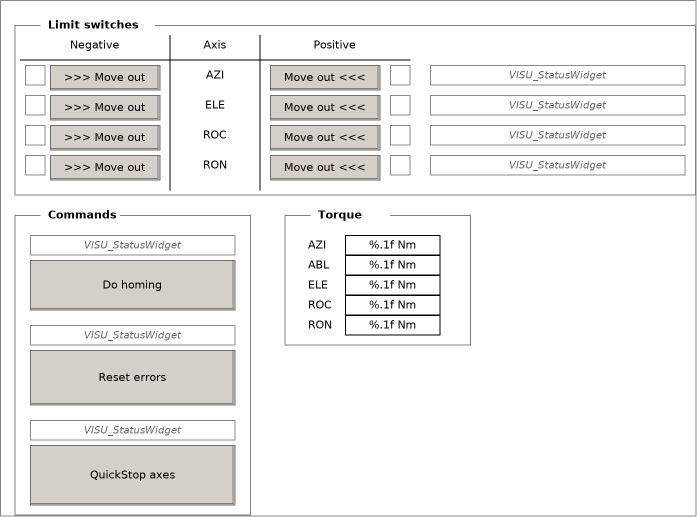
VISUALIZATION VISU_AxesAdvanced  // 697x517
VAR_IN_OUT
	ref : Axes;
    widget : AxesWidget;
END_VAR
    Polyline (120,215) (250,215) (250,515) (15,515) (15,215) (40,215)
    Polyline (155,25) (695,25) (695,195) (15,195) (15,25) (40,25)
    Label (45,15 100x20), "Limit switches"
    Label (170,60 90x30), "AZI"
    Frame (390,65 20x20)
        shows VISU_State_gray_red(state := ref.parts.azi.positiveLimitSwitchError)
    Line (260,190) (260,35)
    Line (170,190) (170,35)
    Label (260,30 150x30), "Positive"
    Label (20,30 150x30), "Negative"
    Line (410,60) (20,60)
    Label (170,30 90x30), "Axis"
    Button (270,65 110x25), "Move out <<<", input disabled if: ref.parts.azi.processes.moveOutOfLimitSwitch.statuses.enabledStatus.disabled
        OnMouseClick: execute { ref.parts.azi.processes.moveOutOfLimitSwitch.set.switch := LimitSwitches.POSITIVE_LIMIT_SWITCH; ref.parts.azi.processes.moveOutOfLimitSwitch.do_request := TRUE; }
    Frame (25,65 20x20)
        shows VISU_State_gray_red(state := ref.parts.azi.negativeLimitSwitchError)
    Button (50,65 110x25), ">>> Move out", input disabled if: ref.parts.azi.processes.moveOutOfLimitSwitch.statuses.enabledStatus.disabled
        OnMouseClick: execute { ref.parts.azi.processes.moveOutOfLimitSwitch.set.switch := LimitSwitches.NEGATIVE_LIMIT_SWITCH; ref.parts.azi.processes.moveOutOfLimitSwitch.do_request := TRUE; }
    Label (170,90 90x30), "ELE"
    Frame (390,95 20x20)
        shows VISU_State_gray_red(state := ref.parts.ele.positiveLimitSwitchError)
    Button (270,95 110x25), "Move out <<<", input disabled if: ref.parts.ele.processes.moveOutOfLimitSwitch.statuses.enabledStatus.disabled
        OnMouseClick: execute { ref.parts.ele.processes.moveOutOfLimitSwitch.set.switch := LimitSwitches.POSITIVE_LIMIT_SWITCH; ref.parts.ele.processes.moveOutOfLimitSwitch.do_request := TRUE; }
    Frame (25,95 20x20)
        shows VISU_State_gray_red(state := ref.parts.ele.negativeLimitSwitchError)
    Button (50,95 110x25), ">>> Move out", input disabled if: ref.parts.ele.processes.moveOutOfLimitSwitch.statuses.enabledStatus.disabled
        OnMouseClick: execute { ref.parts.ele.processes.moveOutOfLimitSwitch.set.switch := LimitSwitches.NEGATIVE_LIMIT_SWITCH; ref.parts.ele.processes.moveOutOfLimitSwitch.do_request := TRUE; }
    Label (170,120 90x30), "ROC"
    Frame (390,125 20x20)
        shows VISU_State_gray_red(state := ref.parts.roc.positiveLimitSwitchError)
    Button (270,125 110x25), "Move out <<<", input disabled if: ref.parts.roc.processes.moveOutOfLimitSwitch.statuses.enabledStatus.disabled
        OnMouseClick: execute { ref.parts.roc.processes.moveOutOfLimitSwitch.set.switch := LimitSwitches.POSITIVE_LIMIT_SWITCH; ref.parts.roc.processes.moveOutOfLimitSwitch.do_request := TRUE; }
    Frame (25,125 20x20)
        shows VISU_State_gray_red(state := ref.parts.roc.negativeLimitSwitchError)
    Button (50,125 110x25), ">>> Move out", input disabled if: ref.parts.roc.processes.moveOutOfLimitSwitch.statuses.enabledStatus.disabled
        OnMouseClick: execute { ref.parts.roc.processes.moveOutOfLimitSwitch.set.switch := LimitSwitches.NEGATIVE_LIMIT_SWITCH; ref.parts.roc.processes.moveOutOfLimitSwitch.do_request := TRUE; }
    Label (170,150 90x30), "RON"
    Frame (390,155 20x20)
        shows VISU_State_gray_red(state := ref.parts.ron.positiveLimitSwitchError)
    Button (270,155 110x25), "Move out <<<", input disabled if: ref.parts.ron.processes.moveOutOfLimitSwitch.statuses.enabledStatus.disabled
        OnMouseClick: execute { ref.parts.ron.processes.moveOutOfLimitSwitch.set.switch := LimitSwitches.POSITIVE_LIMIT_SWITCH; ref.parts.ron.processes.moveOutOfLimitSwitch.do_request := TRUE; }
    Frame (25,155 20x20)
        shows VISU_State_gray_red(state := ref.parts.ron.negativeLimitSwitchError)
    Button (50,155 110x25), ">>> Move out", input disabled if: ref.parts.ron.processes.moveOutOfLimitSwitch.statuses.enabledStatus.disabled
        OnMouseClick: execute { ref.parts.ron.processes.moveOutOfLimitSwitch.set.switch := LimitSwitches.NEGATIVE_LIMIT_SWITCH; ref.parts.ron.processes.moveOutOfLimitSwitch.do_request := TRUE; }
    Frame (430,65 255x20)
        shows VISU_StatusWidget(widget := widget.axes.azi.processes_moveOutOfLimitSwitchStatus)
    Frame (430,95 255x20)
        shows VISU_StatusWidget(widget := widget.axes.ele.processes_moveOutOfLimitSwitchStatus)
    Frame (430,125 255x20)
        shows VISU_StatusWidget(widget := widget.axes.roc.processes_moveOutOfLimitSwitchStatus)
    Frame (430,155 255x20)
        shows VISU_StatusWidget(widget := widget.axes.ron.processes_moveOutOfLimitSwitchStatus)
    Button (30,260 205x50), "Do homing", input disabled if: ref.processes.doHoming.statuses.enabledStatus.disabled
        OnMouseClick: execute { ref.processes.doHoming.do_request := TRUE; }
    Label (45,205 85x20), "Commands"
    Button (30,350 205x55), "Reset errors", input disabled if: ref.processes.reset.statuses.enabledStatus.disabled
        OnMouseClick: execute { ref.processes.reset.do_request := TRUE; }
    Frame (30,325 205x20)
        shows VISU_StatusWidget(widget := widget.processes_resetStatus)
        p4168582468: ref.processes.reset.actualStatus
    Frame (30,235 205x20)
        shows VISU_StatusWidget(widget := widget.processes_doHomingStatus)
        p4168582468: ref.processes.doHoming.actualStatus
    Button (30,445 205x60), "QuickStop axes", input disabled if: ref.processes.quickStop.statuses.enabledStatus.disabled
        OnMouseClick: execute { ref.processes.quickStop.do_request := TRUE; }
    Frame (30,420 205x20)
        shows VISU_StatusWidget(widget := widget.processes_quickStopStatus)
        p4168582468: ref.processes.quickStop.actualStatus
    Label (305,235 40x20), "AZI"
    Rectangle (345,235 95x20), "%.1f Nm", text variable: ref.parts.azi.actTorqueAzi.newtonmeter.value
    Label (305,255 40x20), "ABL"
    Rectangle (345,255 95x20), "%.1f Nm", text variable: ref.parts.azi.actTorqueAbl.newtonmeter.value
    Label (305,275 40x20), "ELE"
    Rectangle (345,275 95x20), "%.1f Nm", text variable: ref.parts.ele.actTorque.newtonmeter.value
    Label (305,295 40x20), "ROC"
    Rectangle (345,295 95x20), "%.1f Nm", text variable: ref.parts.roc.actTorque.newtonmeter.value
    Label (305,315 40x20), "RON"
    Rectangle (345,315 95x20), "%.1f Nm", text variable: ref.parts.ron.actTorque.newtonmeter.value
    Polyline (390,215) (470,215) (470,345) (285,345) (285,215) (310,215)
    Label (315,205 60x20), "Torque"
END_VISUALIZATION

(* stored: Version 1.1.0.1, ProductVersion 3.1.4019.2
   Visu VISU_AxesAdvanced: Id {ec2f8870-7acd-4601-8886-abd94b52237e} *)
